{attribute 'no_check'}
FUNCTION SetOvrVelo : LREAL
VAR_INPUT
	SetVelo													:	LREAL;
	MaxVelo													:	LREAL;
END_VAR
VAR
END_VAR

IF 	MaxVelo = 0.0 
	OR SetVelo = 0.0
THEN
	SetOvrVelo 												:= 0.0;
ELSE                										
	SetOvrVelo 												:= 100.0 / MaxVelo * SetVelo;
END_IF

END_FUNCTION

(* stored: Version 1.1.0.1, ProductVersion 3.1.4024.12
   POU SetOvrVelo: Id {fdae079d-c334-47c4-bf89-4e30fa852178}, SpecialFunc None *)
